PROGRAM ZAxis_Manager
VAR
	ResetError: BOOL;
	
	Offset: LREAL; //general offset of the encoder value
		
	//half the settings have been filled out already. the FB is used to fill the remaining empty variables. fill out the rest of the starting values up here
	VeloOverride: INT := 100; // usually used to slow the motor
	AccOverride: INT := 100; //acceeration or the over ride
	DccOverride: INT := 100; // deceleration of the override
	JerkOverride: INT := 100; //jerk
	ActivateJogFast: BOOL; //trigger for fast movement
	VeloManJog: REAL := 75; //speed of the regular jog movement
	VeloManJogFAST: REAL := 50; // speed of the fast movement
	AccManJOG: REAL := 250; //general ACC
	DccManJog: REAL := 250; // general DCC
	MaxTorque: WORD := 150; //150% of max torque
	
	
//	Forwards  : BOOL;
	ManConsent: BOOL;
//	Backwards  : BOOL;
	Target: INT;
	RefTrigger: BOOL;
	
	ExtraSensorInput: TAxSensorModule; // compressed FUN for exteriour sensor inputs. temp, edge, jog stops
	SpecialOperations: TAxSpecialOperationModule; //compressed FUN for the special operation commands. 
	AxisCoupleIN: TAxCoupleModule; //connects to the AX_Couple_out of the manager from the next axis. NOT MASTER/SLAVE
	Z1_AxisCoupleOUT: TAxCoupleModule; //connects to the AX_Couple_out of the manager from the next axis. NOT MASTER/SLAVE
	Z2_AxisCoupleOUT: TAxCoupleModule; //connects to the AX_Couple_out of the manager from the next axis. NOT MASTER/SLAVE

	DriveIsReal: BOOL; //a check to make sure the drive is real.
	ErrorWordArray: WORD; //build a array of words that act as a cluster of error watching variables. each step in array will be one axis. differant values of the word for each axis mean a differant error. 
	
	ASP: TASPState; //safety interlock system. connects to the safety program OR build a blank ASP that fills all the values but doesnt connect anywhere. 
	
	TargetPositionActivate: BOOL; //starts the drive positing to the Sollpos
	JogStop: LREAL := 1E100 ; // a stopping point using the jog system to signify it is in the right spot. Need to have the LimitPosJOG adjusted after to compensate for the next space.

	
	(*
	//programed commands for movement and controls. NOT part of the PMA build, this is exteriour controls. 
	
	ManVsAutoSW: BOOL;
	ResetButton: BOOL;
	PHYSICALManVsAutoSW: BOOL;
	
	TON_OKdelay: TON;
	*)
	MotorOK: BOOL; // link this into the EL6910 output STO status. then when STO is good this will be good too. 
	
	StartButton: BOOL;
	
	DriveCMD_Z1: DriveCMDShortCUT; //extra system for the FB to make it easy to read.
	DriveCMD_Z2: DriveCMDShortCUT; //extra system for the FB to make it easy to read.
	ASPshortCut_Z1: ASPshortCUT;  // same as above
	ASPshortCut_Z2: ASPshortCUT;  // same as above
	
	ManIN: BOOL;
	AutoIN: BOOL;
	ResetBTN: BOOL;
	SwitchMAN: BOOL;
	SwitchAuto: BOOL;
	AutoRUN: BOOL;
	SafeTEST: BOOL;
	ResetSync: BOOL;
	TOF_ZaxisEnable: TOF;
END_VAR

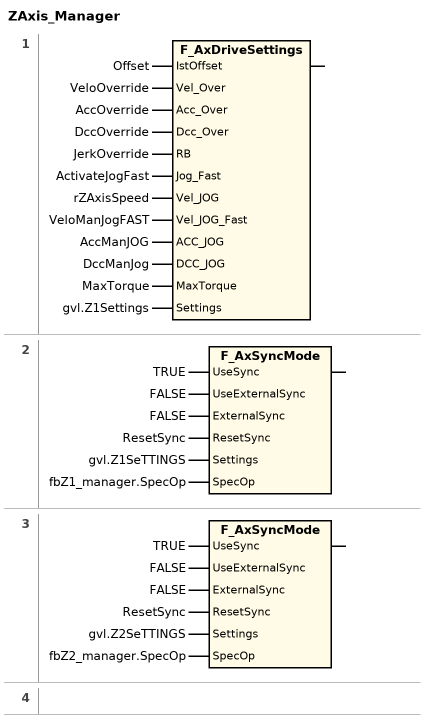
// NETWORK 1
F_AxDriveSettings(IstOffset := Offset, Vel_Over := VeloOverride, Acc_Over := AccOverride, Dcc_Over := DccOverride, RB := JerkOverride, Jog_Fast := ActivateJogFast, Vel_JOG := rZAxisSpeed, Vel_JOG_Fast := VeloManJogFAST, ACC_JOG := AccManJOG, DCC_JOG := DccManJog, MaxTorque := MaxTorque, Settings := gvl.Z1Settings);

// NETWORK 2
F_AxSyncMode(UseSync := TRUE, UseExternalSync := FALSE, ExternalSync := FALSE, ResetSync := ResetSync, Settings := gvl.Z1SeTTINGS, SpecOp := fbZ1_manager.SpecOp);

// NETWORK 3
F_AxSyncMode(UseSync := TRUE, UseExternalSync := FALSE, ExternalSync := FALSE, ResetSync := ResetSync, Settings := gvl.Z2SeTTINGS, SpecOp := fbZ2_manager.SpecOp);

// NETWORK 4

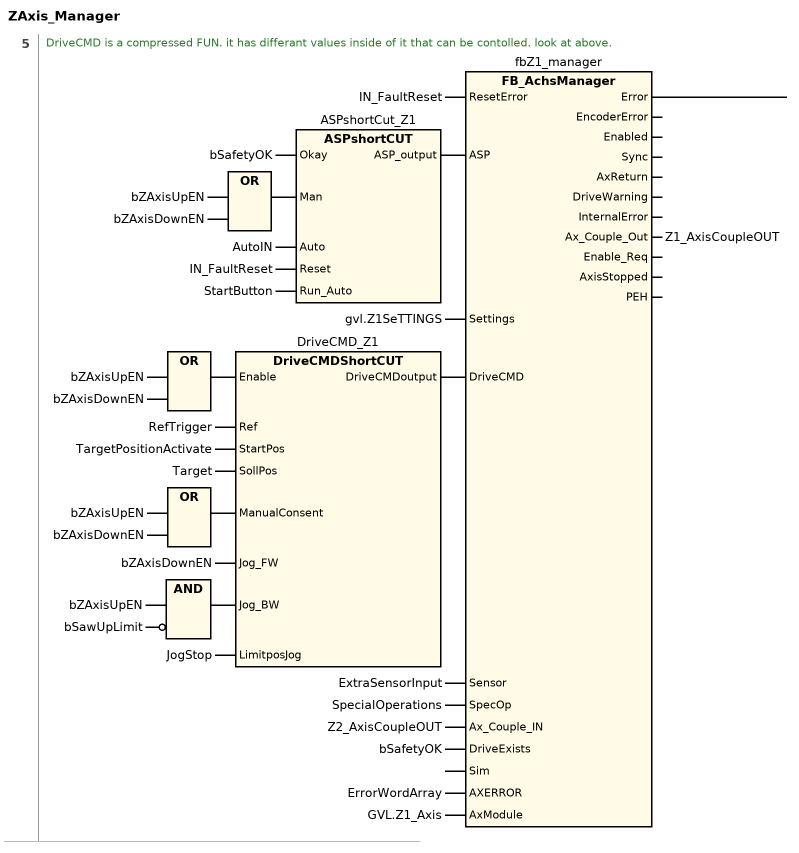
// NETWORK 5
// DriveCMD is a compressed FUN. it has differant values inside of it that can be contolled. look at above.
ASPshortCut_Z1(
    Okay := bSafetyOK,
    Man := bZAxisUpEN OR bZAxisDownEN,
    Auto := AutoIN,
    Reset := IN_FaultReset,
    Run_Auto := StartButton); // ASPshortCUT
DriveCMD_Z1(
    Enable := bZAxisUpEN OR bZAxisDownEN,
    Ref := RefTrigger,
    StartPos := TargetPositionActivate,
    SollPos := Target,
    ManualConsent := bZAxisUpEN OR bZAxisDownEN,
    Jog_FW := bZAxisDownEN,
    Jog_BW := bZAxisUpEN AND NOT bSawUpLimit,
    LimitposJog := JogStop); // DriveCMDShortCUT
fbZ1_manager(
    ResetError := IN_FaultReset,
    ASP := ASPshortCut_Z1.ASP_output,
    Settings := gvl.Z1SeTTINGS,
    DriveCMD := DriveCMD_Z1.DriveCMDoutput,
    Sensor := ExtraSensorInput,
    SpecOp := SpecialOperations,
    Ax_Couple_IN := Z2_AxisCoupleOUT,
    DriveExists := bSafetyOK,
    AXERROR := ErrorWordArray,
    AxModule := GVL.Z1_Axis,
    Ax_Couple_Out => Z1_AxisCoupleOUT); // FB_AchsManager

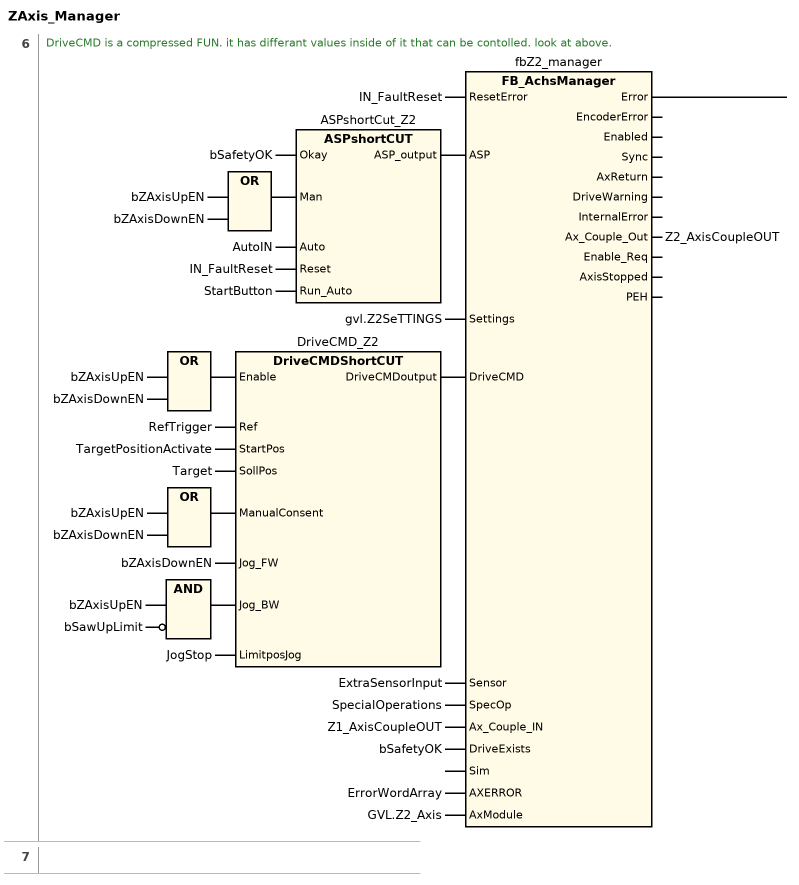
// NETWORK 6
// DriveCMD is a compressed FUN. it has differant values inside of it that can be contolled. look at above.
ASPshortCut_Z2(
    Okay := bSafetyOK,
    Man := bZAxisUpEN OR bZAxisDownEN,
    Auto := AutoIN,
    Reset := IN_FaultReset,
    Run_Auto := StartButton); // ASPshortCUT
DriveCMD_Z2(
    Enable := bZAxisUpEN OR bZAxisDownEN,
    Ref := RefTrigger,
    StartPos := TargetPositionActivate,
    SollPos := Target,
    ManualConsent := bZAxisUpEN OR bZAxisDownEN,
    Jog_FW := bZAxisDownEN,
    Jog_BW := bZAxisUpEN AND NOT bSawUpLimit,
    LimitposJog := JogStop); // DriveCMDShortCUT
fbZ2_manager(
    ResetError := IN_FaultReset,
    ASP := ASPshortCut_Z2.ASP_output,
    Settings := gvl.Z2SeTTINGS,
    DriveCMD := DriveCMD_Z2.DriveCMDoutput,
    Sensor := ExtraSensorInput,
    SpecOp := SpecialOperations,
    Ax_Couple_IN := Z1_AxisCoupleOUT,
    DriveExists := bSafetyOK,
    AXERROR := ErrorWordArray,
    AxModule := GVL.Z2_Axis,
    Ax_Couple_Out => Z2_AxisCoupleOUT); // FB_AchsManager

// NETWORK 7

END_PROGRAM

(* stored: Version 1.1.0.1, ProductVersion 3.1.4024.15
   POU ZAxis_Manager: Id {998db7fd-c2f3-4cfb-bf62-8a82116b63bd}, SpecialFunc None *)
